FUNCTION SinusFunction : REAL
VAR_INPUT
	A : 	REAL; 		//Amplitude
	yoff : 	REAL;		//Offset
	w : 	REAL;		//Kreisfrequenz
	t : 	REAL;		//Zeit
END_VAR
VAR
END_VAR

SinusFunction := A * sin(w*t) + yoff;
RETURN;

END_FUNCTION

(* stored: Version 1.1.0.1, ProductVersion 3.1.4024.13
   POU SinusFunction: Id {df32de09-9cfe-4a68-9b30-a17279fd3013}, SpecialFunc None *)
